// SIMATIC S7-200 project (STEP 7-Micro/WIN), CPU 221 REL 01.10

ORGANIZATION_BLOCK MAIN:OB1
TITLE=PROGRAM COMMENTS
BEGIN
Network 1 // Network Title
// Network Comment
LDN    I0.0
AN     I0.1
LDN    I0.1
AN     I0.2
AN     I0.3
OLD
=      Q0.0
END_ORGANIZATION_BLOCK
